// Mitsubishi GX Works2 project: auto   PLC: Q03UDV

PROGRAM MAIN
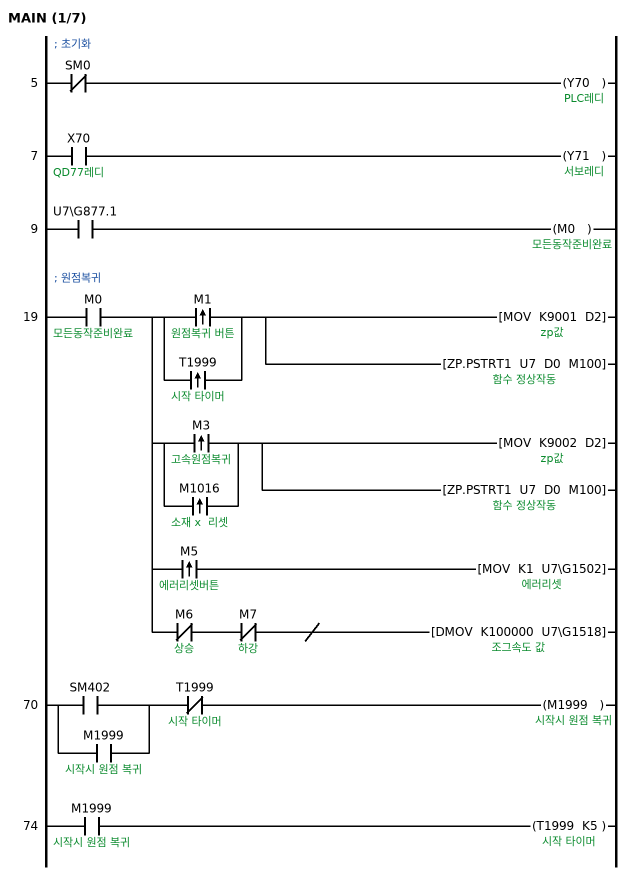
; 초기화
5     LDI     SM0
      OUT     Y70  ; PLC레디
7     LD      X70  ; QD77레디
      OUT     Y71  ; 서보레디
9     LD      U7\G877.1
      OUT     M0  ; 모든동작준비완료
; 원점복귀
19    LD      M0  ; 모든동작준비완료
      MPS
      LDP     M1  ; 원점복귀 버튼
      ORP     T1999  ; 시작 타이머
      ANB
      MOV     K9001 D2  ; zp값
      ZP.PSTRT1 U7 D0 M100  ; 함수 정상작동
      MRD
      LDP     M3  ; 고속원점복귀
      ORP     M1016  ; 소재 x  리셋
      ANB
      MOV     K9002 D2
      ZP.PSTRT1 U7 D0 M100
      MRD
      ANDP    M5  ; 에러리셋버튼
      MOV     K1 U7\G1502  ; 에러리셋
      MPP
      ANI     M6  ; 상승
      ANI     M7  ; 하강
      INV
      DMOV    K100000 U7\G1518  ; 조그속도 값
70    LD      SM402
      OR      M1999  ; 시작시 원점 복귀
      ANI     T1999  ; 시작 타이머
      OUT     M1999  ; 시작시 원점 복귀
74    LD      M1999  ; 시작시 원점 복귀
      OUT     T1999 K5  ; 시작 타이머
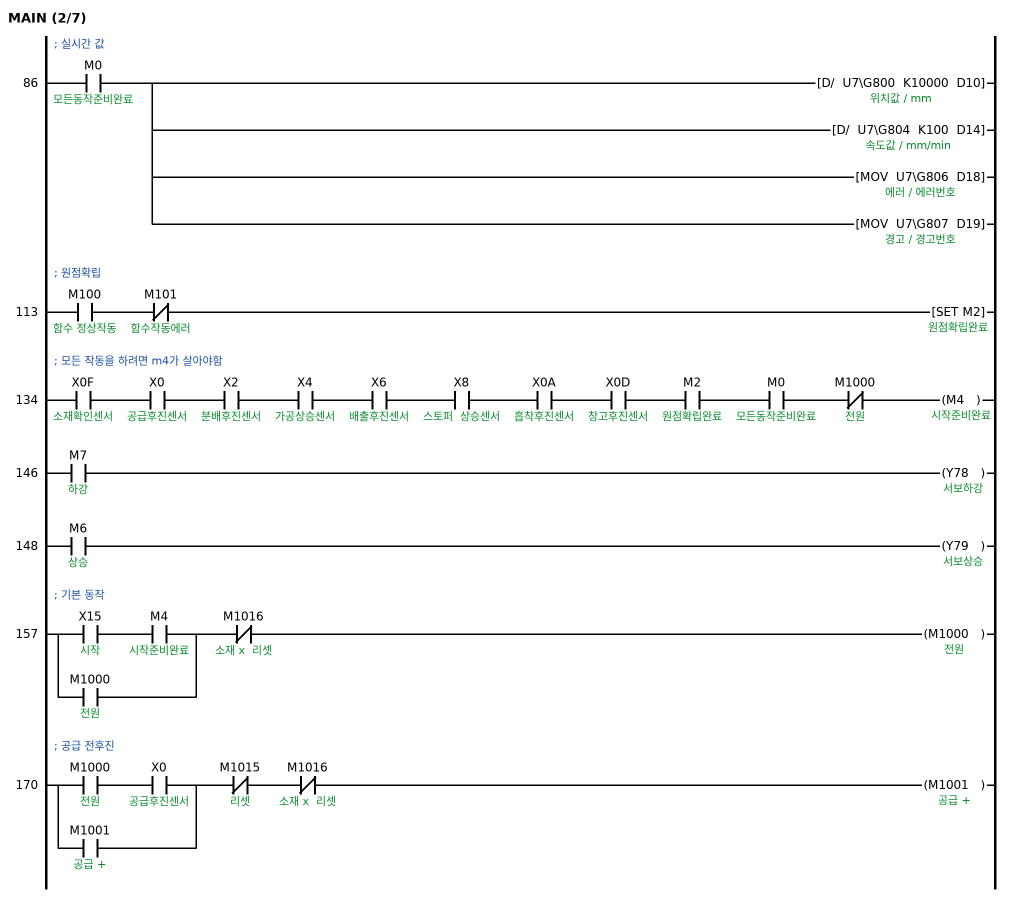
; 실시간 값
86    LD      M0  ; 모든동작준비완료
      D/      U7\G800 K10000 D10  ; 위치값 / mm
      D/      U7\G804 K100 D14  ; 속도값 / mm/min
      MOV     U7\G806 D18  ; 에러 / 에러번호
      MOV     U7\G807 D19  ; 경고 / 경고번호
; 원점확립
113   LD      M100  ; 함수 정상작동
      ANI     M101  ; 함수작동에러
      SET     M2  ; 원점확립완료
; 모든 작동을 하려면 m4가 살아야함
134   LD      X0F  ; 소재확인센서
      AND     X0  ; 공급후진센서
      AND     X2  ; 분배후진센서
      AND     X4  ; 가공상승센서
      AND     X6  ; 배출후진센서
      AND     X8  ; 스토퍼  상승센서
      AND     X0A  ; 흡착후진센서
      AND     X0D  ; 창고후진센서
      AND     M2  ; 원점확립완료
      AND     M0  ; 모든동작준비완료
      ANI     M1000  ; 전원
      OUT     M4  ; 시작준비완료
146   LD      M7  ; 하강
      OUT     Y78  ; 서보하강
148   LD      M6  ; 상승
      OUT     Y79  ; 서보상승
; 기본 동작
157   LD      X15  ; 시작
      AND     M4  ; 시작준비완료
      OR      M1000  ; 전원
      ANI     M1016  ; 소재 x  리셋
      OUT     M1000  ; 전원
; 공급 전후진
170   LD      M1000  ; 전원
      AND     X0  ; 공급후진센서
      OR      M1001  ; 공급 +
      ANI     M1015  ; 리셋
      ANI     M1016  ; 소재 x  리셋
      OUT     M1001  ; 공급 +
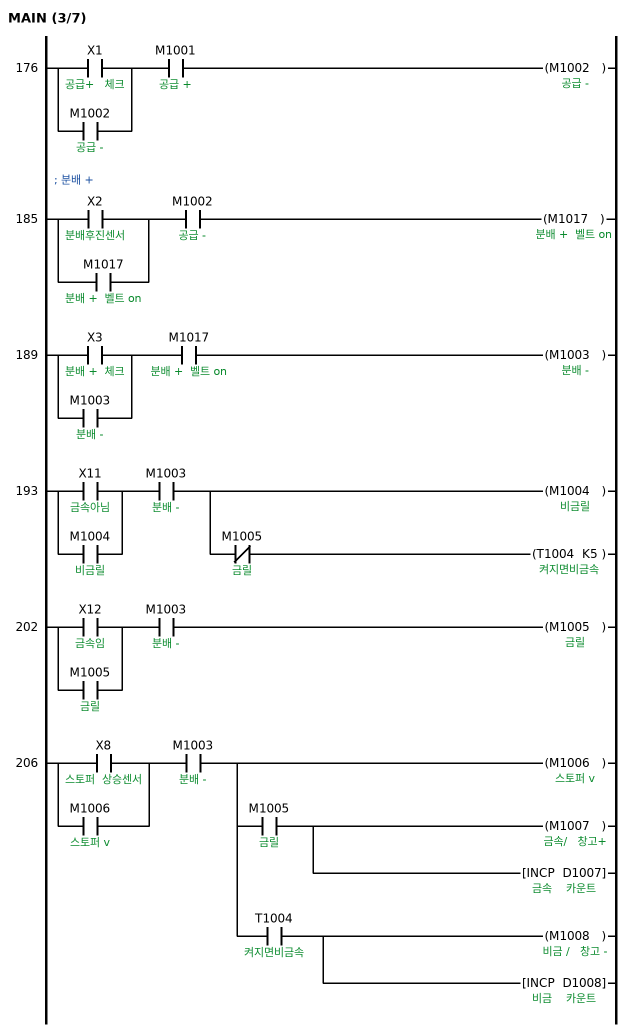
176   LD      X1  ; 공급+   체크
      OR      M1002  ; 공급 -
      AND     M1001  ; 공급 +
      OUT     M1002  ; 공급 -
; 분배 +
185   LD      X2  ; 분배후진센서
      OR      M1017  ; 분배 +  벨트 on
      AND     M1002  ; 공급 -
      OUT     M1017  ; 분배 +  벨트 on
189   LD      X3  ; 분배 +  체크
      OR      M1003  ; 분배 -
      AND     M1017  ; 분배 +  벨트 on
      OUT     M1003  ; 분배 -
193   LD      X11  ; 금속아님
      OR      M1004  ; 비금릴
      AND     M1003  ; 분배 -
      OUT     M1004  ; 비금릴
      ANI     M1005  ; 금릴
      OUT     T1004 K5  ; 켜지면비금속
202   LD      X12  ; 금속임
      OR      M1005  ; 금릴
      AND     M1003  ; 분배 -
      OUT     M1005  ; 금릴
206   LD      X8  ; 스토퍼  상승센서
      OR      M1006  ; 스토퍼 v
      AND     M1003  ; 분배 -
      OUT     M1006  ; 스토퍼 v
      MPS
      AND     M1005  ; 금릴
      OUT     M1007  ; 금속/   창고+
      INCP    D1007  ; 금속    카운트
      MPP
      AND     T1004  ; 켜지면비금속
      OUT     M1008  ; 비금 /   창고 -
      INCP    D1008  ; 비금    카운트
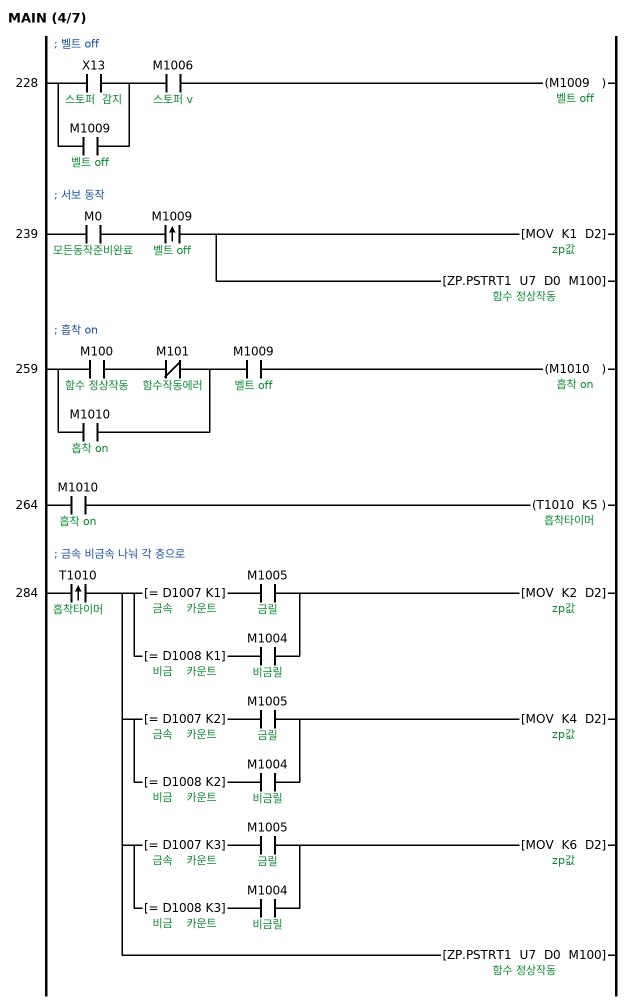
; 벨트 off
228   LD      X13  ; 스토퍼  감지
      OR      M1009  ; 벨트 off
      AND     M1006  ; 스토퍼 v
      OUT     M1009  ; 벨트 off
; 서보 동작
239   LD      M0  ; 모든동작준비완료
      ANDP    M1009  ; 벨트 off
      MOV     K1 D2
      ZP.PSTRT1 U7 D0 M100
; 흡착 on
259   LD      M100  ; 함수 정상작동
      ANI     M101  ; 함수작동에러
      OR      M1010  ; 흡착 on
      AND     M1009  ; 벨트 off
      OUT     M1010  ; 흡착 on
264   LD      M1010  ; 흡착 on
      OUT     T1010 K5  ; 흡착타이머
; 금속 비금속 나눠 각 층으로
284   LDP     T1010  ; 흡착타이머
      MPS
      LD=     D1007 K1  ; 금속    카운트
      AND     M1005  ; 금릴
      LD=     D1008 K1  ; 비금    카운트
      AND     M1004  ; 비금릴
      ORB
      ANB
      MOV     K2 D2
      MRD
      LD=     D1007 K2  ; 금속    카운트
      AND     M1005  ; 금릴
      LD=     D1008 K2  ; 비금    카운트
      AND     M1004  ; 비금릴
      ORB
      ANB
      MOV     K4 D2
      MRD
      LD=     D1007 K3  ; 금속    카운트
      AND     M1005  ; 금릴
      LD=     D1008 K3  ; 비금    카운트
      AND     M1004  ; 비금릴
      ORB
      ANB
      MOV     K6 D2
      MPP
      ZP.PSTRT1 U7 D0 M100
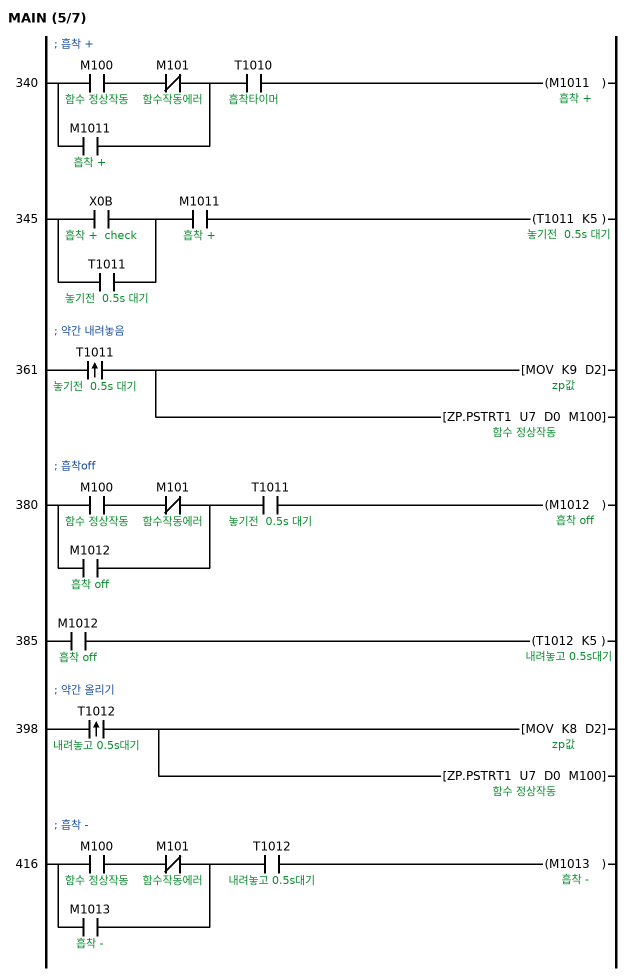
; 흡착 +
340   LD      M100  ; 함수 정상작동
      ANI     M101  ; 함수작동에러
      OR      M1011  ; 흡착 +
      AND     T1010  ; 흡착타이머
      OUT     M1011  ; 흡착 +
345   LD      X0B  ; 흡착 +  check
      OR      T1011  ; 놓기전  0.5s 대기
      AND     M1011  ; 흡착 +
      OUT     T1011 K5  ; 놓기전  0.5s 대기
; 약간 내려놓음
361   LDP     T1011  ; 놓기전  0.5s 대기
      MOV     K9 D2
      ZP.PSTRT1 U7 D0 M100
; 흡착off
380   LD      M100  ; 함수 정상작동
      ANI     M101  ; 함수작동에러
      OR      M1012  ; 흡착 off
      AND     T1011  ; 놓기전  0.5s 대기
      OUT     M1012  ; 흡착 off
385   LD      M1012  ; 흡착 off
      OUT     T1012 K5  ; 내려놓고 0.5s대기
; 약간 올리기
398   LDP     T1012  ; 내려놓고 0.5s대기
      MOV     K8 D2
      ZP.PSTRT1 U7 D0 M100
; 흡착 -
416   LD      M100  ; 함수 정상작동
      ANI     M101  ; 함수작동에러
      OR      M1013  ; 흡착 -
      AND     T1012  ; 내려놓고 0.5s대기
      OUT     M1013  ; 흡착 -
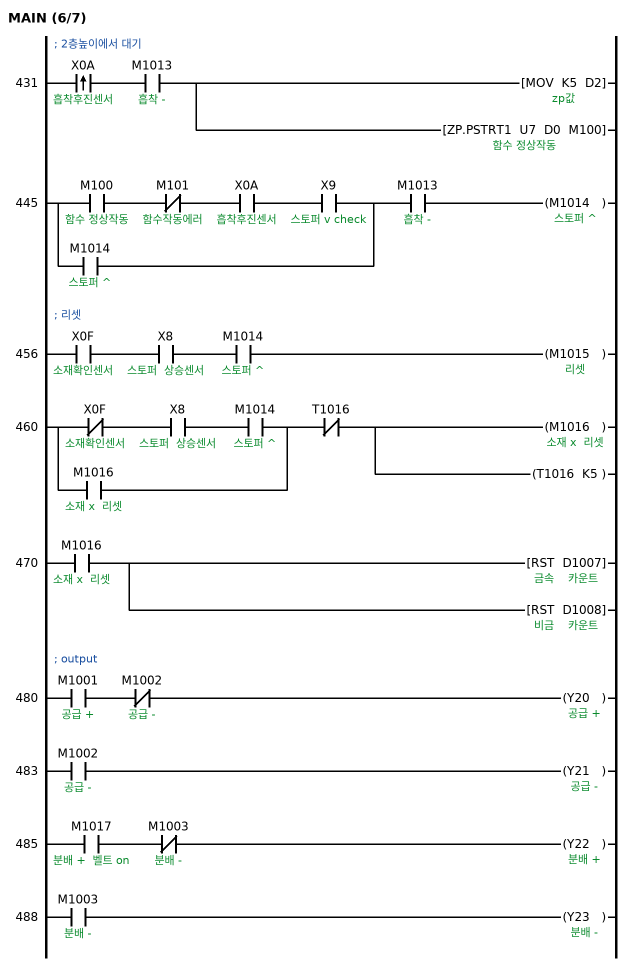
; 2층높이에서 대기
431   LDP     X0A  ; 흡착후진센서
      AND     M1013  ; 흡착 -
      MOV     K5 D2
      ZP.PSTRT1 U7 D0 M100
445   LD      M100  ; 함수 정상작동
      ANI     M101  ; 함수작동에러
      AND     X0A  ; 흡착후진센서
      AND     X9  ; 스토퍼 v check
      OR      M1014  ; 스토퍼 ^
      AND     M1013  ; 흡착 -
      OUT     M1014  ; 스토퍼 ^
; 리셋
456   LD      X0F  ; 소재확인센서
      AND     X8  ; 스토퍼  상승센서
      AND     M1014  ; 스토퍼 ^
      OUT     M1015  ; 리셋
460   LDI     X0F  ; 소재확인센서
      AND     X8  ; 스토퍼  상승센서
      AND     M1014  ; 스토퍼 ^
      OR      M1016  ; 소재 x  리셋
      ANI     T1016
      OUT     M1016  ; 소재 x  리셋
      OUT     T1016 K5
470   LD      M1016  ; 소재 x  리셋
      RST     D1007  ; 금속    카운트
      RST     D1008  ; 비금    카운트
; output
480   LD      M1001  ; 공급 +
      ANI     M1002  ; 공급 -
      OUT     Y20  ; 공급 +
483   LD      M1002  ; 공급 -
      OUT     Y21  ; 공급 -
485   LD      M1017  ; 분배 +  벨트 on
      ANI     M1003  ; 분배 -
      OUT     Y22  ; 분배 +
488   LD      M1003  ; 분배 -
      OUT     Y23  ; 분배 -
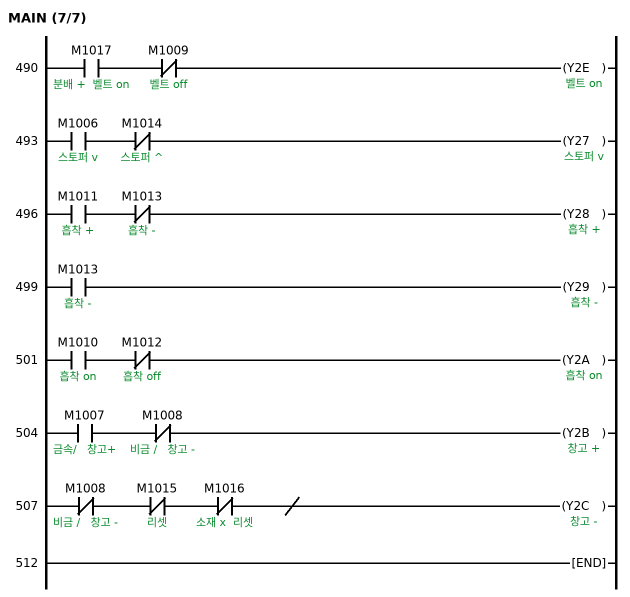
490   LD      M1017  ; 분배 +  벨트 on
      ANI     M1009  ; 벨트 off
      OUT     Y2E  ; 벨트 on
493   LD      M1006  ; 스토퍼 v
      ANI     M1014  ; 스토퍼 ^
      OUT     Y27  ; 스토퍼 v
496   LD      M1011  ; 흡착 +
      ANI     M1013  ; 흡착 -
      OUT     Y28  ; 흡착 +
499   LD      M1013  ; 흡착 -
      OUT     Y29  ; 흡착 -
501   LD      M1010  ; 흡착 on
      ANI     M1012  ; 흡착 off
      OUT     Y2A  ; 흡착 on
504   LD      M1007  ; 금속/   창고+
      ANI     M1008  ; 비금 /   창고 -
      OUT     Y2B  ; 창고 +
507   LDI     M1008  ; 비금 /   창고 -
      ANI     M1015  ; 리셋
      ANI     M1016  ; 소재 x  리셋
      INV
      OUT     Y2C  ; 창고 -
512   END
END_PROGRAM

// device comments not shown above
M1104  ; 분배 -
M1112  ; 흡착 -
T1110  ; 놓기전  0.5초대기
